// TIA Portal V20 export
TYPE "LGM_LKinCtrl_ControlNodeConfig"
// stored: Access Published
   STRUCT
      spare : Bool;
   END_STRUCT;
END_TYPE
